FUNCTION_BLOCK AX_OR_2 (* FB to calculate boolean OR *)
  (* Standard: 61499-2; Description: Copyright (c) 2024 HR Agrartechnik GmbH This program and the accompanying materials are made available under the terms of the Eclipse Public License 2.0 which is available at https://www.eclipse.org/legal/epl-2.0/ SPDX-License-Identifier: EPL-2.0 *)
  (* Version 1.0, 2024-10-23, franz *)
  PACKAGE io::adp::boolean;
  (* Documentation:
  Copyright (c) 2024 HR Agrartechnik GmbH   
   This program and the accompanying materials are made    
   available under the terms of the Eclipse Public License 2.0    
   which is available at https://www.eclipse.org/legal/epl-2.0/    
   SPDX-License-Identifier: EPL-2.0
  *)
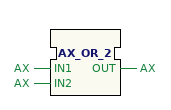
  SOCKETS
    IN1 : AX; (* OR input 1 *)
    IN2 : AX; (* OR input 2 *)
  END_SOCKETS
  PLUGS
    OUT : AX; (* OR result *)
  END_PLUGS
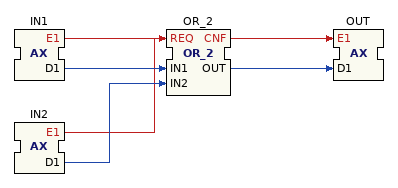
  FBS
    OR_2 : OR_2;
  END_FBS
  EVENT_CONNECTIONS
    IN1.E1 TO OR_2.REQ;
    IN2.E1 TO OR_2.REQ;
    OR_2.CNF TO OUT.E1;
  END_CONNECTIONS
  DATA_CONNECTIONS
    IN1.D1 TO OR_2.IN1;
    IN2.D1 TO OR_2.IN2;
    OR_2.OUT TO OUT.D1;
  END_CONNECTIONS
END_FUNCTION_BLOCK
